{attribute 'linkalways'} 
{attribute 'no_explicit_call' := 'This FB is a CLASS and must be accessed using methods or properties'}
{attribute 'enable_dynamic_creation'}
FUNCTION_BLOCK ABSTRACT NciCommand EXTENDS Command IMPLEMENTS I_NciCommand

END_FUNCTION_BLOCK

(* stored: Version 1.1.0.1, ProductVersion 3.1.4024.12
   POU NciCommand: Id {f023d2d9-2cf2-00e2-37ce-a4781a92b766}, SpecialFunc None *)
